{attribute addProperty BoxType "EK1100-0000-0018"}
{attribute addProperty Id "A_0017_BK1250_0000_0018A_0017_BK1250_0000_0018_9625E6C900"}
{attribute addProperty CRC "1776748706"}
{attribute addProperty SizeInBites "0"}
{attribute addProperty SizeInBytes "0"}
TYPE Term_478_EK1100_69E708A2 EXTENDS EK1100_179A0949 :
STRUCT
	{attribute addProperty Name "A_0017_BK1250_0000_0018"}
	A_0017_BK1250_0000_0018 : A_0017_BK1250_0000_0018_9625E6C9;
END_STRUCT
END_TYPE

(* stored: Version 1.2.0.0, ProductVersion 3.1.4024.9
   DUT Term_478_EK1100_69E708A2: Id {122af385-bc44-4c9a-ba14-814b45ebe706} *)
